Staubli VAL3: Pause.pgx

program Pause(point x_pPoint (dimensions=1))
begin
  movej(appro(x_pPoint,trAppro),tPince,mRapide)
  movel(x_pPoint,tPince,mLent)
  open(tPince)
  movel(appro(x_pPoint,trAppro),tPince,mRapide)
  close(tPince)

end
